(* CODESYS project CtaAppLeistung_1.0.0.6.library
   Description: CtaAppLeistung Library der CTA
   Version: 1.0.0.6
   Title: CtaAppLeistung
   Author: SIS
   Company: CTA
   Placeholder: CtaAppLeistung
   DocFormat: reStructuredText
   DefaultNamespace: CtaAppLeistung
   CompiledLibraryCompatibilityVersion: CODESYS V3.5 SP16 Patch 3
   LanguageModelAttribute: qualified-access-only

Project tree, tasks and I/O mapping:
  libraries: CtaSysConfig, 1.0.0.2 (CTA); CtaAppBasic, 1.0.0.0 (CTA); CtaAppDumper, 1.0.0.0 (CTA); VisuDialogs, * (System); Standard, 3.5.18.0 (System); CtaSysTypes, 1.0.0.0 (CTA); CtaVisSymbols, 1.0.0.0 (CTA); CtaVisHelp, 1.0.0.0 (CTA); VisuSymbols, 4.5.0.0 (System)
  40 Visualizations/
    CONFIG/
      visualisation DIA_CONFIG_HYST_LS_ST
      visualisation VIS_Leistung_Config
    LEISTUNG/
      visualisation DIA_LS_ST
      visualisation VIS_Leistung
  30 Program Organization Units/
    LEISTUNG/
      function block FB_LS_ST [ST]: actConfig
    CONFIG/
      function block FB_CONFIG_HYST_LS_ST [ST]: metGetHystZu, metGetHystWeg, actConfig, proMinHzAkt, proMaxHzAkt, Point, MinHzZu, MinHzWeg, proTHIS, MaxStufen, proRampDelay, proMinStageRuntime
  00000000-0000-0000-0000-000000000000|D:\CoDeSys\LibrariesV3\trunk\Intern\CAA\CAA Template\3.4.0.0 draft\Placeholder.xml
  00000000-0000-0000-0000-000000000000|D:\CoDeSys\LibrariesV3\trunk\Intern\CAA\CAA Template\3.2.0.3 draft\Prefix.pdf
  00000000-0000-0000-0000-000000000000|D:\CoDeSys\LibrariesV3\trunk\Intern\CAA\CAA Template\3.5.2.0 draft\Placeholder.xml
  20 Structs/
    data type scayayPoint
    data type scayMinHzWeg
    data type scayMinHzZu
    data type scHzParameter
    data type scLinePoint
  50 Images/
  10 Documenation/
    global variables VersionHistory
    global variables readMe
  21 Interface/
    CONFIG/
      interface ITF_CONFIG_HYST_LS_ST: metGetHystZu, metGetHystWeg, proMaxHzAkt, proMinHzAkt, MinHzWeg, MinHzZu, Point, proTHIS, MaxStufen, proRampDelay, proMinStageRuntime
  11 Library Parameter/
  12 Konstanten/
    global variables GVL_CONSTANT
  60 Textlisten/
    text list GlobalTextList
    FB_LS_ST/
      text list txtLsStDiagramm
  13 Globale Variablen/
*)

// 20 Structs/scayayPoint
TYPE scayayPoint :
	STRUCT
		ayayPoint : ARRAY[1..GVL_CONSTANT.iMaxArray] OF ARRAY[0..5] OF scLinePoint;
	END_STRUCT
END_TYPE

// 20 Structs/scayMinHzWeg
TYPE scayMinHzWeg :
	STRUCT
		ayMinHzWeg : ARRAY[1..GVL_CONSTANT.iMaxArray] OF REAL;
	END_STRUCT
END_TYPE

// 20 Structs/scayMinHzZu
TYPE scayMinHzZu :
	STRUCT
		ayMinHzZu : ARRAY[1..GVL_CONSTANT.iMaxArray] OF REAL;
	END_STRUCT
END_TYPE

// 20 Structs/scHzParameter
TYPE scHzParameter :
	STRUCT
		rYMinHzAkt  				    :   REAL;                                   // Minimum Hz auf Verdichter Aktueller Betrieb
        rYMaxHzAkt  				    :   REAL;                                   // Maximum Hz auf Verdichter Aktueller Betrieb       
        rYMinHz						    :   REAL;                                   // Minimum Hz auf Verdichter
        rYMaxHz						    :   REAL;                                   // Maximum Hz auf Verdichter
	END_STRUCT
END_TYPE

// 20 Structs/scLinePoint
TYPE scLinePoint :
    STRUCT
        rP1X        :   REAL;
        rP1Y        :   REAL;      
    END_STRUCT
END_TYPE

// 10 Documenation/VersionHistory
(* 

.. image:: ../../Images/CTA_Logo.jpg
   :align: right
   :width: 15% 

**Vorlage**   


============ =========== =========== ============================================
**Date**     **Version** **Author**  **Change**
------------ ----------- ----------- --------------------------------------------
04.03.2021   0.0.0.0     SIS         Vorlage erstellt

============ =========== =========== ============================================


*)
VAR_GLOBAL
    stInfo : STRING:= '0.0.0.0, Vorlage, CTA';
END_VAR

// 10 Documenation/readMe
(*
|	Bibliothek CtaAppLesitung zur Erzeugung des Leistungssignals und der Stufenzuschaltung der Maschine
|	Instanzieren Sie den CtaAppLesitung.FB_LS_ST in ihrem Funktionsbaustein oder POU beispielsweise als fbLeistung.
|	Instanzieren Sie den CtaAppLesitung.FB_CONFIG_HYST_LS_ST in ihrem Funktionsbaustein oder POU beispielsweise als fbLeistungConfig.
|	Deklarieren Sie die Struktur Variable welche als Parameter und zur ansteuerung dienen wie im Code beispiel.
|  
| *Beispiel* 

+-----------------------+---------------------------------------------------------------------------------------------------------------------------------------------------------------------------------------------------------------------------------------------------------------------------------------------------------------------------------------------------------------------------------------------------------------------------------------+
| Beschreibung          |  Code                                                                                                                                                                                                                                                                                                                                                                                                                                 |
+=======================+=======================================================================================================================================================================================================================================================================================================================================================================================================================================+
| Pou oder SmFb         | .. code-block:: codesys                                                                                                                                                                                                                                                                                                                                                                                                               |
|                       |                                                                                                                                                                                                                                                                                                                                                                                                                                       |
|                       |	// Deklaration als VAR im POU oder dem selbsterstellten Funktionsbaustein                                                                                                                                                                                                                                                                                                                                                       	|
|                       |   VAR   																																																																																																								|
|						|	    (*Einsatzgrenze Verdichter1*)																																																		 																																															|
|						|		fbLeistung			: CtaAppVerdichter.FB_LS_ST;                                                                                                                                                                                                                                                                                                                                                              					|
|						|		fbLeistungConfig	: CtaAppVerdichter.FB_CONFIG_HYST_LS_ST;                                                                                                                                                                                                                                                                                                                                                            		|
| 						|	END_VAR                                                                                                                                                                                                                                                                                                                                                                                                                         	|
+-----------------------+---------------------------------------------------------------------------------------------------------------------------------------------------------------------------------------------------------------------------------------------------------------------------------------------------------------------------------------------------------------------------------------------------------------------------------------+
| Code für Init         | .. code-block:: codesys                                                                                                                                                                                                                                                                                                                                                                                                               |
|                       |   																																																																																																									|
| 						|	// Kopieren des nachfolgenden Codes in eine Action zur Initialisierung der Parameter. Zum Beispiel actConfig.																																																																														|
|                       |	{region "Parameter Einsatzgrenzen Verdichter1"}                                                                                                                                                                                                                                                                                                                                                                                     |
|						|		fbLeistung.fbrMinHzFu            								   		(_wertInit :=  30.0				, _minInit :=		, _maxInit :=		);		//P1 Diagrammgrösse Y Achse Max																																																											|
|						|		fbLeistung.fbrMaxHzFu													(_wertInit :=  50.0				, _minInit :=		, _maxInit :=		);		//P2 Diagrammgrösse Y Achse Min																																																											|
|						|	{endregion}																																																		 																																																					|
|                       |	{region "Parameter Einsatzgrenzen Verdichter1"}                                                                                                                                                                                                                                                                                                                                                                                     |
|						|		fbLeistungConfig.fbrMinHzAktLimit            							(_wertInit :=  30.0				, _minInit :=		, _maxInit :=		);		//P1 Diagrammgrösse Y Achse Max																																																											|
|						|		fbLeistungConfig.fbrMaxHzAktLimit										(_wertInit :=  50.0				, _minInit :=		, _maxInit :=		);		//P2 Diagrammgrösse Y Achse Min																																																											|
|						|		fbLeistungConfig.fbusiMaxStufen            								(_wertInit :=   4.0				, _minInit :=		, _maxInit :=		);		//P1 Diagrammgrösse Y Achse Max																																																											|
|						|		fbLeistungConfig.fbtRampDelay											(_wertInit :=  T#1M				, _minInit :=		, _maxInit :=		);		//P2 Diagrammgrösse Y Achse Min																																																											|
|						|		fbLeistungConfig.fbtMinStageRuntime            							(_wertInit :=  T#1M				, _minInit :=		, _maxInit :=		);		//P1 Diagrammgrösse Y Achse Max																																																											|
|						|	{endregion}																																																		 																																																					|
+-----------------------+---------------------------------------------------------------------------------------------------------------------------------------------------------------------------------------------------------------------------------------------------------------------------------------------------------------------------------------------------------------------------------------------------------------------------------------+
*)                                                                                                                                                                                                                                                                                                                                                                                                                                                              
 VAR_GLOBAL                                                                                                                                                                                                                                                                                                                                                                                                                                                      
    xReadMeDone              :   BOOL;                                                                                                                                                                                                                                                                                                                                                                                                                           
END_VAR

// 12 Konstanten/GVL_CONSTANT
{attribute 'qualified_only'}
VAR_GLOBAL CONSTANT
	iMaxArray				:	INT	:= 16;	
END_VAR

// 21 Interface/CONFIG/ITF_CONFIG_HYST_LS_ST
INTERFACE ITF_CONFIG_HYST_LS_ST EXTENDS __System.IQueryinterface

METHOD metGetHystZu : REAL
VAR_INPUT
	iPos	:	INT;
END_VAR
END_METHOD

METHOD metGetHystWeg : REAL
VAR_INPUT
	iPos	:	INT;
END_VAR
END_METHOD

PROPERTY proMaxHzAkt : REAL
GET
END_GET
END_PROPERTY

PROPERTY proMinHzAkt : REAL
GET
END_GET
END_PROPERTY

PROPERTY MinHzWeg : REFERENCE TO ARRAY[1..GVL_CONSTANT.iMaxArray] OF REAL;
GET
END_GET
END_PROPERTY

PROPERTY MinHzZu : REFERENCE TO ARRAY[1..GVL_CONSTANT.iMaxArray] OF REAL;
GET
END_GET
END_PROPERTY

PROPERTY Point : REFERENCE TO ARRAY[1..GVL_CONSTANT.iMaxArray] OF ARRAY[0..5] OF scLinePoint;
GET
END_GET
END_PROPERTY

PROPERTY proTHIS : REFERENCE TO FB_CONFIG_HYST_LS_ST
GET
END_GET
END_PROPERTY

PROPERTY MaxStufen : USINT
GET
END_GET
END_PROPERTY

PROPERTY proRampDelay : TIME
GET
END_GET
END_PROPERTY

PROPERTY proMinStageRuntime : TIME
GET
END_GET
END_PROPERTY

END_INTERFACE

// 30 Program Organization Units/CONFIG/FB_CONFIG_HYST_LS_ST
FUNCTION_BLOCK FB_CONFIG_HYST_LS_ST IMPLEMENTS ITF_CONFIG_HYST_LS_ST
VAR_INPUT
	rMinHzAkt				:	REAL	:= 30;
	rMaxHzAkt				:	REAL	:= 70;	
END_VAR
VAR_OUTPUT
END_VAR
VAR
	iFor				:	INT;
	ayItffbrHystZu 		: 	ARRAY[1..GVL_CONSTANT.iMaxArray] OF CtaSysConfig.ITF_REAL;
	ayItffbrHystWeg		: 	ARRAY[1..GVL_CONSTANT.iMaxArray] OF CtaSysConfig.ITF_REAL;	
	ayayPoint 			: 	ARRAY[1..GVL_CONSTANT.iMaxArray] OF ARRAY[0..5] OF scLinePoint;
	ayMinHzWeg 			: 	ARRAY[1..GVL_CONSTANT.iMaxArray] OF REAL;
	ayMinHzZu 			: 	ARRAY[1..GVL_CONSTANT.iMaxArray] OF REAL;
	
	(* CONFIG *)    	
	fbConfigFile		:	CtaSysConfig.fbConfigFile;
	fbrMinHzAktLimit	:	CtaSysConfig.fbREAL;
	fbrMaxHzAktLimit	:	CtaSysConfig.fbREAL;
	fbusiMaxStufen		:	CtaSysConfig.fbUSINT;
	fbtRampDelay		:	CtaSysConfig.fbTIME;
	fbtMinStageRuntime	:	CtaSysConfig.fbTIME;
	fbConfigFile1		:	CtaSysConfig.fbConfigFile;
	ayfbrHystZu			:	ARRAY[1..GVL_CONSTANT.iMaxArray] OF CtaSysConfig.fbREAL;
	fbConfigFile2		:	CtaSysConfig.fbConfigFile;
	ayfbrHystWeg		:	ARRAY[1..GVL_CONSTANT.iMaxArray] OF CtaSysConfig.fbREAL;
END_VAR

// (* Config *)
// Activate configuration settings
actConfig();

// (* Begrenzung *)
// Limits the values of rMinHzAkt and rMaxHzAkt within specified min and max limits
rMinHzAkt := LIMIT(fbrMinHzAktLimit.rValue, rMinHzAkt, fbrMaxHzAktLimit.rValue);
rMaxHzAkt := LIMIT(fbrMinHzAktLimit.rValue, rMaxHzAkt, fbrMaxHzAktLimit.rValue);

// (* Min hz zu *)
// Sets the minimum threshold values (ayMinHzZu) for each array element up to the maximum defined in iMaxArray
FOR iFor := 1 TO GVL_CONSTANT.iMaxArray DO
    ayMinHzZu[iFor] := ((rMinHzAkt * iFor) + metGetHystZu(iFor));
END_FOR;

// (* Min Hz Weg *)
// Limits and assigns values to the array ayMinHzWeg based on the minimum threshold and array element values, ensuring each element is one less than the corresponding value in ayMinHzZu
FOR iFor := 1 TO GVL_CONSTANT.iMaxArray DO
    ayMinHzWeg[iFor] := LIMIT(0, ((rMinHzAkt * iFor) + metGetHystWeg(iFor) + metGetHystZu(iFor)), ayMinHzZu[iFor] - 1);
END_FOR;

// (* ayayPoint *)
// Defines coordinates for points based on scaling factors and limits for each array element within iMaxArray
FOR iFor := 1 TO GVL_CONSTANT.iMaxArray DO
    // Checks if current step (usiValue) is within the maximum defined
    IF fbusiMaxStufen.usiValue >= iFor THEN
        // Calculate coordinates for points based on scaled values and limits
        ayayPoint[iFor][0].rP1X := CtaAppBasic.fcScale(ayMinHzZu[iFor], ayMinHzZu[1], MAX((fbusiMaxStufen.usiValue + 1) * rMinHzAkt,fbusiMaxStufen.usiValue * rMaxHzAkt), 0, 100);
        ayayPoint[iFor][0].rP1y := 0;

        ayayPoint[iFor][1].rP1X := CtaAppBasic.fcScale(ayMinHzZu[iFor], ayMinHzZu[1],  MAX((fbusiMaxStufen.usiValue + 1) * rMinHzAkt,fbusiMaxStufen.usiValue * rMaxHzAkt), 0, 100);
        ayayPoint[iFor][1].rP1y := LIMIT(rMinHzAkt, ayMinHzZu[iFor] / iFor, rMaxHzAkt);

        ayayPoint[iFor][2].rP1X := CtaAppBasic.fcScale(MAX(rMinHzAkt * iFor, ayMinHzZu[iFor]), ayMinHzZu[1], MAX((fbusiMaxStufen.usiValue + 1) * rMinHzAkt,fbusiMaxStufen.usiValue * rMaxHzAkt), 0, 100);
        ayayPoint[iFor][2].rP1y := LIMIT(rMinHzAkt, ayMinHzZu[iFor] / iFor, rMaxHzAkt);

        // Conditional to check if the next threshold exceeds max frequency limit
        IF ayMinHzZu[iFor + 1] >= rMaxHzAkt * iFor AND iFor + 1 <= fbusiMaxStufen.usiValue THEN
            ayayPoint[iFor][3].rP1X := CtaAppBasic.fcScale(rMaxHzAkt * iFor, ayMinHzZu[1],  MAX((fbusiMaxStufen.usiValue + 1) * rMinHzAkt,fbusiMaxStufen.usiValue * rMaxHzAkt), 0, 100);
            ayayPoint[iFor][3].rP1y := rMaxHzAkt;
            ayayPoint[iFor][4].rP1X := SEL(iFor = fbusiMaxStufen.usiValue, CtaAppBasic.fcScale(ayMinHzZu[iFor + 1], ayMinHzZu[1],  MAX((fbusiMaxStufen.usiValue + 1) * rMinHzAkt,fbusiMaxStufen.usiValue * rMaxHzAkt), 0, 100), 100);
            ayayPoint[iFor][4].rP1y := rMaxHzAkt;
        ELSE
            ayayPoint[iFor][3].rP1X := SEL(iFor = fbusiMaxStufen.usiValue, CtaAppBasic.fcScale(ayMinHzZu[iFor + 1], ayMinHzZu[1],  MAX((fbusiMaxStufen.usiValue + 1) * rMinHzAkt,fbusiMaxStufen.usiValue * rMaxHzAkt), 0, 100), 100);
            ayayPoint[iFor][3].rP1y := LIMIT(rMinHzAkt, CtaAppBasic.fcScale(ayayPoint[iFor][3].rP1X, 0, 100, rMinHzAkt,  MAX((fbusiMaxStufen.usiValue + 1) * rMinHzAkt,fbusiMaxStufen.usiValue * rMaxHzAkt)) / iFor, rMaxHzAkt);
            ayayPoint[iFor][4].rP1X := ayayPoint[iFor][3].rP1X;
            ayayPoint[iFor][4].rP1y := ayayPoint[iFor][3].rP1y;
        END_IF;

        // Assign values for final point based on max threshold and current step
        ayayPoint[iFor][5].rP1X := ayayPoint[iFor][4].rP1X;
        ayayPoint[iFor][5].rP1y := SEL(iFor = fbusiMaxStufen.usiValue, LIMIT(rMinHzAkt, ayMinHzZu[iFor + 1] / (iFor + 1), rMaxHzAkt), 0);
    ELSE
        // Set default zero values for points if step exceeds max allowed value
        ayayPoint[iFor][0].rP1X := 0;
        ayayPoint[iFor][0].rP1y := 0;
        ayayPoint[iFor][1].rP1X := 0;
        ayayPoint[iFor][1].rP1y := 0;
        ayayPoint[iFor][2].rP1X := 0;
        ayayPoint[iFor][2].rP1y := 0;
        ayayPoint[iFor][3].rP1X := 0;
        ayayPoint[iFor][3].rP1y := 0;
        ayayPoint[iFor][4].rP1X := 0;
        ayayPoint[iFor][4].rP1y := 0;
        ayayPoint[iFor][5].rP1X := 0;
        ayayPoint[iFor][5].rP1y := 0;
    END_IF;
END_FOR;

METHOD metGetHystZu : REAL
VAR_INPUT
	iPos	:	INT;
END_VAR
IF iPos >= TO_INT(LOWER_BOUND(ayfbrHystzu,1)) AND iPos <= TO_INT(UPPER_BOUND(ayfbrHystzu,1)) THEN
	metGetHystZu := ayfbrHystzu[iPos].rValue;
ELSE
	metGetHystZu := 0;
END_IF;
END_METHOD

METHOD metGetHystWeg : REAL
VAR_INPUT
	iPos	:	INT;
END_VAR
IF iPos >= TO_INT(LOWER_BOUND(ayfbrHystWeg,1)) AND iPos <= TO_INT(UPPER_BOUND(ayfbrHystWeg,1)) THEN
	metGetHystWeg := ayfbrHystWeg[iPos].rValue;
ELSE
	metGetHystWeg := 0;
END_IF;
END_METHOD

ACTION actConfig:
(* ConfigFile *)
fbConfigFile();
fbrMinHzAktLimit	(_usiParaNr := 1,itfConfigFb := fbConfigFile);
fbrMaxHzAktLimit	(_usiParaNr := 2,itfConfigFb := fbConfigFile);
fbusiMaxStufen		(_usiParaNr := 3,itfConfigFb := fbConfigFile,_MinInit := 1,_maxInit := 16);
fbtRampDelay		(_usiParaNr := 4,itfConfigFb := fbConfigFile,_MinInit := T#10S,_maxInit := T#49D);
fbtMinStageRuntime	(_usiParaNr := 5,itfConfigFb := fbConfigFile,_MinInit := T#10S,_maxInit := T#49D);

IF fbrMinHzAktLimit.proStateChanged THEN
	rMinHzAkt := fbrMinHzAktLimit.proValue;
END_IF;

IF fbrMaxHzAktLimit.proStateChanged THEN
	rMaxHzAkt := fbrMaxHZAktLimit.proValue;
END_IF;

(* ConfigFile *)
fbConfigFile1();
(* Zuschalt Hysterese *)
FOR iFor := 1 TO GVL_CONSTANT.iMaxArray DO 
	ayfbrHystZu[iFor](_usiParaNr := TO_USINT(iFor+1),itfConfigFb := fbConfigFile1);
	ayItffbrHystZu[iFor] := ayfbrHystZu[iFor];
END_FOR;

(* ConfigFile *)
fbConfigFile2();
(* Wegschalt Hysterese *)
FOR iFor := 1 TO GVL_CONSTANT.iMaxArray DO 
	ayfbrHystWeg[iFor](_usiParaNr := TO_USINT(iFor),itfConfigFb := fbConfigFile2);
	ayItffbrHystWeg[iFor] := ayfbrHystWeg[iFor];
END_FOR;
END_ACTION

PROPERTY proMinHzAkt : REAL
GET
proMinHzAkt := LIMIT(fbrMinHzAktLimit.rValue,rMinHzAkt,fbrMaxHzAktLimit.rValue);
END_GET
END_PROPERTY

PROPERTY proMaxHzAkt : REAL
GET
proMaxHzAkt := LIMIT(fbrMinHzAktLimit.rValue,rMaxHzAkt,fbrMaxHzAktLimit.rValue);
END_GET
END_PROPERTY

PROPERTY Point : REFERENCE TO ARRAY[1..GVL_CONSTANT.iMaxArray] OF ARRAY[0..5] OF scLinePoint;
GET
Point REF= ayayPoint;
END_GET
END_PROPERTY

PROPERTY MinHzZu : REFERENCE TO ARRAY[1..GVL_CONSTANT.iMaxArray] OF REAL;
GET
VAR
	iForayMinHzZu : INT;
END_VAR
MinHzZu REF= ayMinHzZu;
END_GET
END_PROPERTY

PROPERTY MinHzWeg : REFERENCE TO ARRAY[1..GVL_CONSTANT.iMaxArray] OF REAL;
GET
VAR
	iForayMinHzWeg	:	INT;
END_VAR
MinHzWeg REF= ayMinHzWeg;
END_GET
END_PROPERTY

PROPERTY proTHIS : REFERENCE TO FB_CONFIG_HYST_LS_ST
GET
proTHIS REF= THIS^;
END_GET
END_PROPERTY

PROPERTY MaxStufen : USINT
GET
MaxStufen := fbusiMaxStufen.usiValue;
END_GET
END_PROPERTY

PROPERTY proRampDelay : TIME
GET
proRampDelay := fbtRampDelay.tValue;
END_GET
END_PROPERTY

PROPERTY proMinStageRuntime : TIME
GET
proMinStageRuntime	:= fbtMinStageRuntime.tValue;
END_GET
END_PROPERTY

END_FUNCTION_BLOCK

// 30 Program Organization Units/LEISTUNG/FB_LS_ST
FUNCTION_BLOCK FB_LS_ST
VAR_INPUT
	xRelease					:   BOOL;
	rRelease					:   REAL;
	iAcknowledge				:   INT;
	ITF_CONFIG_HYST_LS_ST_IN	:	ITF_CONFIG_HYST_LS_ST;		
END_VAR         			
VAR_OUTPUT      			
	iStufen						:	INT;
	rDemande					:	REAL;
	scHz						:	CtaSysTypes.scHzParameter;
END_VAR         			
VAR             			
	ayayPoint					:	ARRAY[1..GVL_CONSTANT.iMaxArray] OF ARRAY[0..5] OF scLinePoint;
	aySoll						:	ARRAY[0..0] OF scLinePoint;
	ayMinHzZu					:	ARRAY[1..GVL_CONSTANT.iMaxArray] OF REAL;
	ayMinHzWeg					:	ARRAY[1..GVL_CONSTANT.iMaxArray] OF REAL;
	iRepaint					:	int;
	iFor						:	INT;
	fbDumpRelease				:	CtaAppDumper.fbDumper;
	fbDumpMinHz					:	CtaAppDumper.fbDumper;
	fbDumpMaxHz					:	CtaAppDumper.fbDumper;
	fbDumpDemand				:	CtaAppDumper.fbDumper;
	(* CONFIG *)
	fbConfigFile				:	CtaSysConfig.fbConfigFile;	
	fbrMinHzFu					:	CtaSysConfig.fbREAL;
	fbrMaxHzFu					:	CtaSysConfig.fbREAL;
	
	iAcknowledgeOld				:	INT;
	iStufenOld					:	INT;
	
	tRampenZuschaltDelay		:	TIME;
	tStufenWegschaltDelay		:	TIME;
	
	TP_RampenZuschaltDelay		:	Standard.TP;	
	TP_StufenWegschaltDelay		:	Standard.TP;
END_VAR

(* Config *)
//actConfig(); Exeption?
(* ConfigFile *)
fbConfigFile();

fbrMinHzFu		(_usiParaNr := 1,itfConfigFb := fbConfigFile,_MinInit := 0,_MaxInit := 200);
fbrMaxHzFu		(_usiParaNr := 2,itfConfigFb := fbConfigFile,_MinInit := 0,_MaxInit := 200);


rRelease := LIMIT(0,rRelease,100);

fbDumpRelease(	xEn 	:=	xRelease,
				rSoll	:=	rRelease,
				rY		=> 	rRelease);
				
IF fbConfigFile.proInitDone THEN
	(* Check Interface *)
	IF __QUERYINTERFACE(ITF_CONFIG_HYST_LS_ST_IN,ITF_CONFIG_HYST_LS_ST_IN) THEN	
		ayMinHzZu				:= ITF_CONFIG_HYST_LS_ST_IN.MinHzZu;
		ayMinHzWeg				:= ITF_CONFIG_HYST_LS_ST_IN.MinHzWeg;
		ayayPoint 				:= ITF_CONFIG_HYST_LS_ST_IN.Point;
		tRampenZuschaltDelay	:= ITF_CONFIG_HYST_LS_ST_IN.proRampDelay;
		tStufenWegschaltDelay	:=	ITF_CONFIG_HYST_LS_ST_IN.proMinStageRuntime;
		(* Stufen & Leistung *)	
		IF xRelease THEN				
			iStufen := MAX(1,iStufen);
			IF iStufen < ITF_CONFIG_HYST_LS_ST_IN.MaxStufen AND CtaAppBasic.fcScale(ayMinHzZu[iStufen+1],ayMinHzZu[1],MAX((ITF_CONFIG_HYST_LS_ST_IN.MaxStufen + 1)*ITF_CONFIG_HYST_LS_ST_IN.proMinHzAkt,ITF_CONFIG_HYST_LS_ST_IN.MaxStufen*ITF_CONFIG_HYST_LS_ST_IN.proMaxHzAkt),0,100) <= rRelease THEN
				iStufen := iStufen + 1;
			ELSIF CtaAppBasic.fcScale(ayMinHzWeg[iStufen],ayMinHzZu[1],MAX((ITF_CONFIG_HYST_LS_ST_IN.MaxStufen + 1)*ITF_CONFIG_HYST_LS_ST_IN.proMinHzAkt,ITF_CONFIG_HYST_LS_ST_IN.MaxStufen*ITF_CONFIG_HYST_LS_ST_IN.proMaxHzAkt),0,100) >= rRelease OR iStufen > ITF_CONFIG_HYST_LS_ST_IN.MaxStufen THEN
				rRelease := CtaAppBasic.fcScale(ayMinHzWeg[iStufen],ayMinHzZu[1],MAX((ITF_CONFIG_HYST_LS_ST_IN.MaxStufen + 1)*ITF_CONFIG_HYST_LS_ST_IN.proMinHzAkt,ITF_CONFIG_HYST_LS_ST_IN.MaxStufen*ITF_CONFIG_HYST_LS_ST_IN.proMaxHzAkt),0,100);	 // änderung durch SIS für langsames retour fahren vor abschaltung
				IF NOT TP_StufenWegschaltDelay.Q AND (rDemande <= 1 OR iAcknowledge < iStufen) THEN				
					iStufen := iStufen - 1;
				END_IF;
			END_IF;			
			(* Soll *)
			aySoll[0].rP1X := rRelease;
			aySoll[0].rP1Y := LIMIT(scHz.rYMinHz,LIMIT(ITF_CONFIG_HYST_LS_ST_IN.proMinHzAkt,CtaAppBasic.fcScale(CtaAppBasic.fcScale(rRelease,SEL(MAX(1,iStufen) = 1,ayayPoint[MAX(1,iStufen)-1][5].rP1X,0),ayayPoint[MAX(1,iStufen)][5].rP1X,0,100,),0,100, ayMinHzZu[MAX(1,iStufen)]/MAX(1,iStufen),CtaAppBasic.fcScale(ayayPoint[MAX(1,iStufen)][5].rP1X,0,100,ITF_CONFIG_HYST_LS_ST_IN.proMinHzAkt,MAX((ITF_CONFIG_HYST_LS_ST_IN.MaxStufen + 1)*ITF_CONFIG_HYST_LS_ST_IN.proMinHzAkt,ITF_CONFIG_HYST_LS_ST_IN.MaxStufen*ITF_CONFIG_HYST_LS_ST_IN.proMaxHzAkt))/MAX(1,iStufen)),ITF_CONFIG_HYST_LS_ST_IN.proMaxHzAkt),scHz.rYMaxHz);
		ELSE
			rRelease 		:= 0;
			iStufen  		:= 0;
			aySoll[0].rP1X	:= 0;
			aySoll[0].rP1Y	:= 0;
		END_IF;
	ELSE
		rRelease 		:= 0;
		iStufen  		:= 0;
		aySoll[0].rP1X	:= 0;
		aySoll[0].rP1Y	:= 0;
		tRampenZuschaltDelay	:= 	T#1M;
		tStufenWegschaltDelay	:=	T#1M;
		FOR iFor := 0 TO GVL_CONSTANT.iMaxArray DO
			ayayPoint[iFor][0].rP1X := 0;
			ayayPoint[iFor][0].rP1Y := 0;
			ayayPoint[iFor][1].rP1X := 0;
			ayayPoint[iFor][1].rP1Y := 0;
			ayayPoint[iFor][2].rP1X := 0;
			ayayPoint[iFor][2].rP1Y := 0;
			ayayPoint[iFor][3].rP1X := 0;
			ayayPoint[iFor][3].rP1Y := 0;
			ayayPoint[iFor][4].rP1X := 0;
			ayayPoint[iFor][4].rP1Y := 0;
			ayayPoint[iFor][5].rP1X := 0;
			ayayPoint[iFor][5].rP1Y := 0;
		END_FOR;
	END_IF;
END_IF;
IF __QUERYINTERFACE(ITF_CONFIG_HYST_LS_ST_IN,ITF_CONFIG_HYST_LS_ST_IN) THEN
	fbDumpDemand(	xEn 	:= xRelease AND NOT TP_RampenZuschaltDelay.Q,
					rSoll 	:= LIMIT(	0,
										CtaAppBasic.fcScale(rIn 	:= 	SEL(xRelease AND NOT TP_RampenZuschaltDelay.Q, 0, rRelease),
															rMin	:= 	SEL(MAX(1,iAcknowledge) = 1,ayayPoint[MAX(1,iAcknowledge)-1][4].rP1X,0),
															rMax	:=	ayayPoint[MAX(1,iAcknowledge)][3].rP1X,
															rOutMin	:=	0,
															rOutMax :=	CtaAppBasic.fcScale(rIn	 	:= ayayPoint[MAX(1,iAcknowledge)][3].rP1Y,
																							rMin 	:= ITF_CONFIG_HYST_LS_ST_IN.proMinHzAkt,
																							rMax 	:= ITF_CONFIG_HYST_LS_ST_IN.proMaxHzAkt,
																							rOutMin	:= 0,
																							rOutMax	:= 100)),
										100),
					rY 		=> rDemande);
ELSE
	rDemande := 0;
END_IF;
// Rampenverzögerung von rDemand bei Zu oder Wegschaltung von Stufen
TP_RampenZuschaltDelay(	IN := iAcknowledge > iAcknowledgeOld,
						PT := tRampenZuschaltDelay);
						
IF TP_RampenZuschaltDelay.Q THEN	
	rDemande := 0;
END_IF

TP_StufenWegschaltDelay(IN := iStufen > iStufenOld,
						PT := tStufenWegschaltDelay	);

scHz.rYMinHz 		:= fbrMinHzFu.rValue;
scHz.rYMaxHz 		:= fbrMaxHzFu.rValue;
fbDumpMinHz.rSoll 	:= ayMinHzZu[MAX(1,iAcknowledge)]/MAX(1,iAcknowledge);
fbDumpMinHz(xEn 	:= xRelease,
			rY		 => scHz.rYMinHzAkt);
IF __QUERYINTERFACE(ITF_CONFIG_HYST_LS_ST_IN,ITF_CONFIG_HYST_LS_ST_IN) THEN
	fbDumpMaxHz.rSoll := ITF_CONFIG_HYST_LS_ST_IN.proMaxHzAkt;
	
ELSE
	fbDumpMaxHz.rSoll := 0;
END_IF;
fbDumpMaxHz(xEn 	:= xRelease,
			rY 		=> scHz.rYMaxHzAkt);	
				
ITF_CONFIG_HYST_LS_ST_IN := 0;

iStufenOld := iStufen;
iAcknowledgeOld := iAcknowledge;

IF iRepaint < 1000 THEN
	iRepaint := iRepaint + 1;
ELSE
	iRepaint := 0;
END_IF;

ACTION actConfig:
(* ConfigFile *)
fbConfigFile();

(*Dumper*)
fbDumpRelease.scParameter.fbrTup		(_WertInit	:=	0.1 ,	_MinInit := ,	_MaxInit :=	);
fbDumpRelease.scParameter.fbrTdown		(_WertInit	:= 	0.1	,	_MinInit := ,	_MaxInit :=	);
fbDumpRelease.scParameter.fbrBand		(_WertInit	:= 50.0	, 	_MinInit := ,	_MaxInit :=	);
fbDumpRelease.scParameter.fbxInExpOut	(_WertInit := FALSE);

fbDumpMinHz.scParameter.fbrTup			(_WertInit	:=	0.1 ,	_MinInit := ,	_MaxInit :=	);
fbDumpMinHz.scParameter.fbrTdown		(_WertInit	:= 	0.1	,	_MinInit := ,	_MaxInit :=	);
fbDumpMinHz.scParameter.fbrBand			(_WertInit	:= 50.0	, 	_MinInit := ,	_MaxInit :=	);
fbDumpMinHz.scParameter.fbxInExpOut		(_WertInit := FALSE);

fbDumpMaxHz.scParameter.fbrTup			(_WertInit	:=	0.1 ,	_MinInit := ,	_MaxInit :=	);
fbDumpMaxHz.scParameter.fbrTdown		(_WertInit	:= 	0.1	,	_MinInit := ,	_MaxInit :=	);
fbDumpMaxHz.scParameter.fbrBand			(_WertInit	:= 50.0	, 	_MinInit := ,	_MaxInit :=	);
fbDumpMaxHz.scParameter.fbxInExpOut		(_WertInit := FALSE);

fbDumpDemand.scParameter.fbrTup			(_WertInit	:=	0.1 ,	_MinInit := ,	_MaxInit :=	);
fbDumpDemand.scParameter.fbrTdown		(_WertInit	:= 	0.1	,	_MinInit := ,	_MaxInit :=	);
fbDumpDemand.scParameter.fbrBand		(_WertInit	:= 50.0	, 	_MinInit := ,	_MaxInit :=	);
fbDumpDemand.scParameter.fbxInExpOut	(_WertInit := FALSE);

fbrMinHzFu		(_usiParaNr := 1,itfConfigFb := fbConfigFile,_MinInit := 0,_MaxInit := 200);
fbrMaxHzFu		(_usiParaNr := 2,itfConfigFb := fbConfigFile,_MinInit := 0,_MaxInit := 200);
END_ACTION

END_FUNCTION_BLOCK

// 40 Visualizations/CONFIG/DIA_CONFIG_HYST_LS_ST
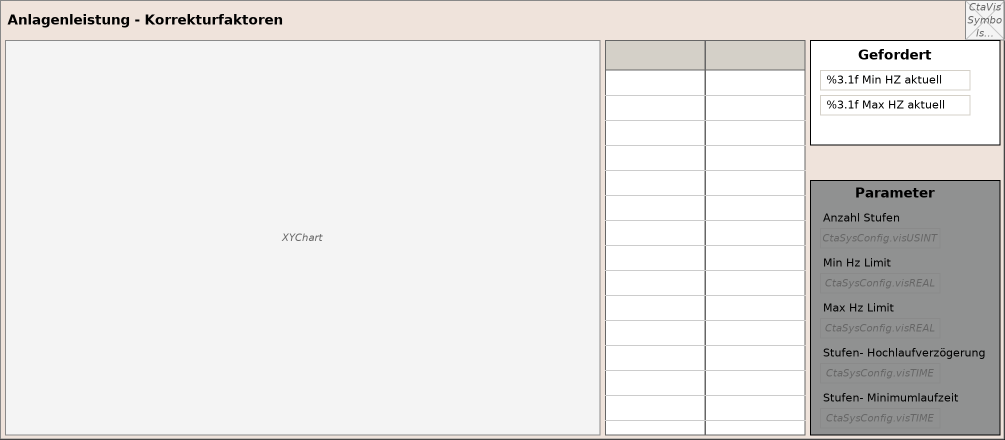
VISUALIZATION DIA_CONFIG_HYST_LS_ST  // 1005x440
VAR_IN_OUT
	{attribute 'VAR_IN_OUT_AS_POINTER'}
	FB_CONFIG_HYST_LS_ST_IN	:	FB_CONFIG_HYST_LS_ST;	
END_VAR
    Rectangle (0,0 1005x440)
    Image (965,0 40x40), image: CtaVisSymbols.ImagePool.close_solo_black
        OnMouseClick:  Dialog=Current Dialog, Result=None, NumpadKeypadSet=True
    Label (0,0 232x40), "Anlagenleistung - Korrekturfaktoren"
    Table (605,40 100x395), data array: FB_CONFIG_HYST_LS_ST_IN.ayItffbrHystZu
        p1014161805: GVL_CONSTANT.iMaxArray - 1 + INT#1
        p208337472: %s HZ
        p3854506369: FB_CONFIG_HYST_LS_ST_IN.ayItffbrHystZu[INDEX].proMax
        p1892666644: FB_CONFIG_HYST_LS_ST_IN.ayItffbrHystZu[INDEX].proMin
        p338671338: FB_CONFIG_HYST_LS_ST_IN.ayItffbrHystZu[INDEX].proValue
        p2170511999: FB_CONFIG_HYST_LS_ST_IN.ayItffbrHystZu[INDEX].proIsLoading
        p3723444502: FB_CONFIG_HYST_LS_ST_IN.ayItffbrHystZu[INDEX].proIsSaving
        p1218418051: FB_CONFIG_HYST_LS_ST_IN.ayItffbrHystZu[INDEX].proParaNr
        p746581629: FB_CONFIG_HYST_LS_ST_IN.ayItffbrHystZu[INDEX].proSaveOnChange
        p3104783080: FB_CONFIG_HYST_LS_ST_IN.ayItffbrHystZu[INDEX].proShowValue
        p2501879983: FB_CONFIG_HYST_LS_ST_IN.ayItffbrHystZu[INDEX].proStrPara
        p1128707560: FB_CONFIG_HYST_LS_ST_IN.fbusiMaxStufen.usiValue
        Columns.Column.[2].Template: OnMouseClick: write the text variable via Default
    Table (705,40 100x395), data array: FB_CONFIG_HYST_LS_ST_IN.ayItffbrHystWeg
        p208337472: %s HZ
        p3854506369: FB_CONFIG_HYST_LS_ST_IN.ayItffbrHystWeg[INDEX].proMax
        p1892666644: FB_CONFIG_HYST_LS_ST_IN.ayItffbrHystWeg[INDEX].proMin
        p338671338: FB_CONFIG_HYST_LS_ST_IN.ayItffbrHystWeg[INDEX].proValue
        p2170511999: FB_CONFIG_HYST_LS_ST_IN.ayItffbrHystWeg[INDEX].proIsLoading
        p3723444502: FB_CONFIG_HYST_LS_ST_IN.ayItffbrHystWeg[INDEX].proIsSaving
        p1218418051: FB_CONFIG_HYST_LS_ST_IN.ayItffbrHystWeg[INDEX].proParaNr
        p746581629: FB_CONFIG_HYST_LS_ST_IN.ayItffbrHystWeg[INDEX].proSaveOnChange
        p3104783080: FB_CONFIG_HYST_LS_ST_IN.ayItffbrHystWeg[INDEX].proShowValue
        p2501879983: FB_CONFIG_HYST_LS_ST_IN.ayItffbrHystWeg[INDEX].proStrPara
        p7306298: FB_CONFIG_HYST_LS_ST_IN.ayfbrHystWeg[INDEX].proMax
        p1933151965: FB_CONFIG_HYST_LS_ST_IN.ayfbrHystWeg[INDEX].proMin
        p3863566920: FB_CONFIG_HYST_LS_ST_IN.ayfbrHystWeg[INDEX].proShowValue
        p2192122294: FB_CONFIG_HYST_LS_ST_IN.ayfbrHystWeg[INDEX].proStrPara
        p400160035: FB_CONFIG_HYST_LS_ST_IN.ayfbrHystWeg[INDEX].proValue
        p1265227338: FB_CONFIG_HYST_LS_ST_IN.ayfbrHystWeg[INDEX]._usiParaNr
        p3726181087: FB_CONFIG_HYST_LS_ST_IN.ayfbrHystWeg[INDEX].itfConfigFb
        p3136911649: FB_CONFIG_HYST_LS_ST_IN.ayfbrHystWeg[INDEX].scState
        p797552052: FB_CONFIG_HYST_LS_ST_IN.ayfbrHystWeg[INDEX].itfConfigFbSync
        p60375027: FB_CONFIG_HYST_LS_ST_IN.ayfbrHystWeg[INDEX].proIsLoading
        p2531912550: FB_CONFIG_HYST_LS_ST_IN.ayfbrHystWeg[INDEX].proIsSaving
        p693678525: FB_CONFIG_HYST_LS_ST_IN.ayfbrHystWeg[INDEX].proParaNr
        p3156763944: FB_CONFIG_HYST_LS_ST_IN.ayfbrHystWeg[INDEX].proSaveOnChange
        p1014161805: GVL_CONSTANT.iMaxArray - 1 + INT#1
        p1128707560: FB_CONFIG_HYST_LS_ST_IN.fbusiMaxStufen.usiValue
        Columns.Column.[2].Template: OnMouseClick: write the text variable via Default
    Rectangle (810,180 190x255)
    Label (820,183 150x20), "Parameter"
    Label (820,253 150x20), "Min Hz Limit"
    Label (820,298 150x20), "Max Hz Limit"
    Frame (820,318 120x20)
        shows CtaSysConfig.visREAL(visfbREALIn := FB_CONFIG_HYST_LS_ST_IN.fbrMaxHzAktLimit, stPhysikalischeEinheit := 'HZ')
    Frame (820,273 120x20)
        shows CtaSysConfig.visREAL(visfbREALIn := FB_CONFIG_HYST_LS_ST_IN.fbrMinHzAktLimit, stPhysikalischeEinheit := 'HZ')
    XYChart (5,40 595x395)
    Frame (820,228 120x20)
        shows CtaSysConfig.visUSINT(visfbUSINTIn := FB_CONFIG_HYST_LS_ST_IN.fbusiMaxStufen)
    Label (820,208 150x20), "Anzahl Stufen"
    Rectangle (810,40 190x105)
    Textfield (820,70 150x20), "%3.1f Min HZ aktuell", text variable: FB_CONFIG_HYST_LS_ST_IN.rMinHzAkt
    Textfield (820,95 150x20), "%3.1f Max HZ aktuell", text variable: FB_CONFIG_HYST_LS_ST_IN.rMaxHzAkt
    Label (820,45 150x20), "Gefordert"
    Label (820,343 170x20), "Stufen- Hochlaufverzögerung"
    Frame (820,363 120x20)
        shows CtaSysConfig.visTIME(visfbTIMEIn := FB_CONFIG_HYST_LS_ST_IN.fbtRampDelay)
    Label (820,388 175x20), "Stufen- Minimumlaufzeit"
    Frame (820,408 120x20)
        shows CtaSysConfig.visTIME(visfbTIMEIn := FB_CONFIG_HYST_LS_ST_IN.fbtMinStageRuntime)
END_VISUALIZATION

// 40 Visualizations/LEISTUNG/DIA_LS_ST
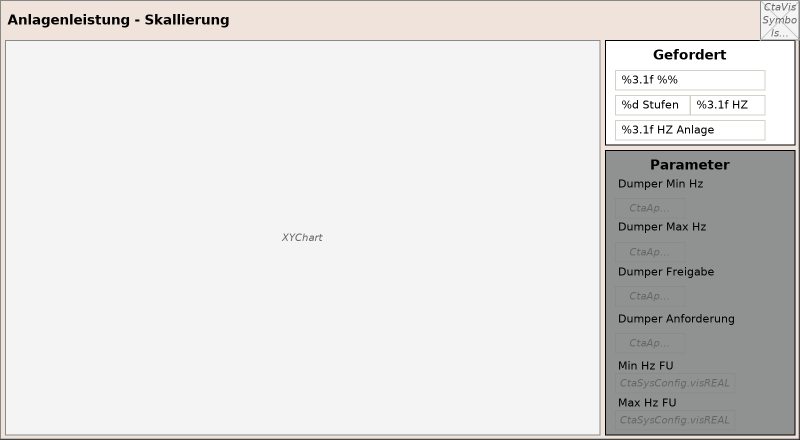
VISUALIZATION DIA_LS_ST  // 800x440
VAR_IN_OUT
	{attribute 'VAR_IN_OUT_AS_POINTER'}
	FB_LS_ST_IN	:	FB_LS_ST;	
END_VAR
    Rectangle (0,0 800x440)
    Rectangle (605,150 190x285)
    Rectangle (605,40 190x105)
    XYChart (5,40 595x395)
    Textfield (615,70 150x20), "%3.1f %%", text variable: FB_LS_ST_IN.aySoll[0].rP1X
    Textfield (690,95 75x20), "%3.1f HZ", text variable: FB_LS_ST_IN.aySoll[0].rP1Y
    Textfield (615,95 75x20), "%d Stufen", text variable: FB_LS_ST_IN.iStufen
    Label (615,45 150x20), "Gefordert"
    Label (615,155 150x20), "Parameter"
    Frame (615,373 120x20)
        shows CtaSysConfig.visREAL(visfbREALIn := FB_LS_ST_IN.fbrMinHzFu, stPhysikalischeEinheit := 'HZ')
    Label (615,356 150x20), "Min Hz FU"
    Label (615,393 150x20), "Max Hz FU"
    Frame (615,410 120x20)
        shows CtaSysConfig.visREAL(visfbREALIn := FB_LS_ST_IN.fbrMaxHzFu, stPhysikalischeEinheit := 'HZ')
    Image (760,0 40x40), image: CtaVisSymbols.ImagePool.close_solo_black
        OnMouseClick:  Dialog=Current Dialog, Result=None, NumpadKeypadSet=True
    Label (0,0 200x40), "Anlagenleistung - Skallierung"
    Textfield (615,120 150x20), "%3.1f HZ Anlage", text variable: FB_LS_ST_IN.aySoll[0].rP1Y* FB_LS_ST_IN.iStufen
    Label (615,174 150x20), "Dumper Min Hz"
    Label (615,217 150x20), "Dumper Max Hz"
    Label (615,262 150x20), "Dumper Freigabe"
    Frame (615,286 70x20)
        shows CtaAppDumper.visDumper(fbDumper := FB_LS_ST_IN.fbDumpRelease)
    Frame (615,242 70x20)
        shows CtaAppDumper.visDumper(fbDumper := FB_LS_ST_IN.fbDumpMaxHz)
    Frame (615,198 70x20)
        shows CtaAppDumper.visDumper(fbDumper := FB_LS_ST_IN.fbDumpMinHz)
    Label (615,309 150x20), "Dumper Anforderung"
    Frame (615,333 70x20)
        shows CtaAppDumper.visDumper(fbDumper := FB_LS_ST_IN.fbDumpDemand)
END_VISUALIZATION

// 40 Visualizations/LEISTUNG/VIS_Leistung
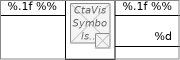
VISUALIZATION VIS_Leistung  // 180x60
VAR_IN_OUT
	FB_LS_ST		:	FB_LS_ST;
END_VAR
    Line (75,46) (180,46)
    Textfield (0,0 60x13), "%.1f %%", text variable: FB_LS_ST.rRelease
    Line (0,15) (180,15)
    Textfield (115,0 60x13), "%.1f %%", text variable: FB_LS_ST.rDemande
    Group (65,0 50x60)
        OnMouseDown:  Dialog=DIA_LS_ST, Parameters={FB_LS_ST_IN: FB_LS_ST}, Selected={0: }, OpenCentered=True
        Textfield (0,0 50x60)
        Image (5,3 40x40), image: CtaVisSymbols.ImagePool.Chart
        Image (30,33 15x15), image: CtaVisSymbols.ImagePool.SettingsSmall
    Textfield (115,30 60x13), "%d", text variable: FB_LS_ST.iStufen
END_VISUALIZATION

// 40 Visualizations/CONFIG/VIS_Leistung_Config
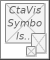
VISUALIZATION VIS_Leistung_Config  // 50x60
VAR_IN_OUT
	FB_CONFIG_HYST_LS_ST	:	FB_CONFIG_HYST_LS_ST;
END_VAR
    Group (0,0 50x60)
        OnMouseClick:  Dialog=DIA_CONFIG_HYST_LS_ST, Parameters={FB_CONFIG_HYST_LS_ST_IN: FB_CONFIG_HYST_LS_ST}, Selected={0: }, OpenCentered=True
        Textfield (0,0 50x60)
        Image (5,3 40x40), image: CtaVisSymbols.ImagePool.Chart
        Image (31,33 15x20), image: CtaVisSymbols.ImagePool.FileDescription
        Image (26,46 10x10), image: CtaVisSymbols.ImagePool.SettingsSmall
END_VISUALIZATION

(* text list txtLsStDiagramm (id | default)
  Hz | Hz
  % | %
   |  *)
